TYPE RudongPump_IOData_1 :
STRUCT
	///泵头型号(0-8)
	O_PumpType: INT;
	///软管型号
	O_HosePipeType: INT;
END_STRUCT
END_TYPE

(* stored: Version 1.1.0.1, ProductVersion 3.1.4024.9
   DUT RudongPump_IOData_1: Id {03679625-ca6c-4978-bb05-dae853ce2b2f} *)
